(* PLC project marvel_telescope, Institute of Astronomy Onto 0.0.1 *)
(* stored: creationDateTime 2025-01-01T00:00:00.0, modificationDateTime 2025-01-01T00:00:00.0 *)

{attribute 'qualified_only'}
TYPE TelescopeNasmythPort : (UNKNOWN := 0, CHANGING := 1, POS_1 := 2, POS_2 := 3) BYTE;
END_TYPE

TYPE TelescopeProcesses : STRUCT
  {attribute 'TcHmiSymbol.Show'}
  initialize : Process;  (* Start initializing *)
  {attribute 'TcHmiSymbol.Show'}
  lock : Process;  (* Lock the cover *)
  {attribute 'TcHmiSymbol.Show'}
  unlock : Process;  (* Unlock the cover *)
  {attribute 'TcHmiSymbol.Show'}
  changeOperatingState : ChangeOperatingStateProcess;  (* Change the operating state (e.g. AUTO, MANUAL, ...) *)
  {attribute 'TcHmiSymbol.Show'}
  slewToCoordinates : PointAlphaDeltaProcess;  (* Slew to the given equatorial coordinates *)
  {attribute 'TcHmiSymbol.Show'}
  slewToAziEle : TelescopeSlewToAziEleProcess;  (* Slew to the given horizontal coordinates *)
  {attribute 'TcHmiSymbol.Show'}
  syncToCoordinates : PointAlphaDeltaProcess;  (* Sync to the given equatorial coordinates *)
  {attribute 'TcHmiSymbol.Show'}
  syncToAziEle : TelescopeSlewToAziEleProcess;  (* Sync to the given horizontal coordinates *)
  {attribute 'TcHmiSymbol.Show'}
  syncToTarget : Process;  (* Sync to the given target *)
  {attribute 'TcHmiSymbol.Show'}
  selectNasmythPort : TelescopeSelectNasmythPortProcess;  (* Select a nasmyth port *)
  {attribute 'TcHmiSymbol.Show'}
  abortSlew : Process;  (* Stop the slewing *)
  {attribute 'TcHmiSymbol.Show'}
  reset : Process;  (* Reset any errors *)
  {attribute 'TcHmiSymbol.Show'}
  powerOn : Process;  (* Power on the axes *)
  {attribute 'TcHmiSymbol.Show'}
  powerOff : Process;  (* Power off the axes *)
  {attribute 'TcHmiSymbol.Show'}
  moveKnownPosition : TelescopeMoveKnownPositionProcess;  (* Move the telescope to the given known position *)
  {attribute 'TcHmiSymbol.Show'}
  setTracking : TelescopeSetTrackingProcess;  (* Power on the axes *)
  {attribute 'TcHmiSymbol.Show'}
  moveM2 : TelescopeMoveProcess;  (* Move M2 to the given position in mm *)
  {attribute 'TcHmiSymbol.Show'}
  openCover : Process;  (* Open the telescope cover *)
  {attribute 'TcHmiSymbol.Show'}
  closeCover : Process;  (* Close the telescope cover *)
  {attribute 'TcHmiSymbol.Show'}
  pulseGuide : TelescopePulseGuideProcess;  (* Pulse guide *)
  {attribute 'TcHmiSymbol.Show'}
  guideRateAlpha : TelescopeSetRateProcess;  (* Guide right ascention rate *)
  {attribute 'TcHmiSymbol.Show'}
  guideRateDelta : TelescopeSetRateProcess;  (* Guide declination rate *)
END_STRUCT;
END_TYPE

TYPE TelescopeStatuses : STRUCT
  {attribute 'OPC.UA.DA' := '1'}
  {attribute 'OPC.UA.DA.Access' := '1'}
  {attribute 'TcHmiSymbol.Show'}
  init : InitializationStatus;
  {attribute 'OPC.UA.DA' := '1'}
  {attribute 'OPC.UA.DA.Access' := '1'}
  {attribute 'TcHmiSymbol.Show'}
  health : HealthStatus;
  {attribute 'OPC.UA.DA' := '1'}
  {attribute 'OPC.UA.DA.Access' := '1'}
  {attribute 'TcHmiSymbol.Show'}
  busy : BusyStatus;
  {attribute 'OPC.UA.DA' := '1'}
  {attribute 'OPC.UA.DA.Access' := '1'}
  {attribute 'TcHmiSymbol.Show'}
  operating : OperatingStatus;
  {attribute 'OPC.UA.DA' := '1'}
  {attribute 'OPC.UA.DA.Access' := '1'}
  {attribute 'TcHmiSymbol.Show'}
  powered : PoweredStatus;
END_STRUCT;
END_TYPE

TYPE TelescopeKnownPositionConfig : STRUCT
  {attribute 'TcHmiSymbol.Show'}
  name : STRING;  (* The name of the position (e.g. 'PARK') *)
  {attribute 'TcHmiSymbol.Show'}
  allowObserver : BOOL;  (* Can an observer switch to this position? *)
  {attribute 'TcHmiSymbol.Show'}
  azi : LREAL;  (* Azimuth in degrees *)
  {attribute 'TcHmiSymbol.Show'}
  ele : LREAL;  (* Elevation in degrees *)
  {attribute 'TcHmiSymbol.Show'}
  rot : LREAL;  (* Nasmyth rotation in degrees *)
  {attribute 'TcHmiSymbol.Show'}
  doAzi : BOOL;  (* Change the azimuth axis to the 'azi' position *)
  {attribute 'TcHmiSymbol.Show'}
  doEle : BOOL;  (* Change the elevation axis to the 'ele' position *)
  {attribute 'TcHmiSymbol.Show'}
  doRot : BOOL;  (* Change the nasmyth rotation axis to the 'rot' position *)
END_STRUCT;
END_TYPE

TYPE TelescopeKnownPositionsConfig : STRUCT
  {attribute 'TcHmiSymbol.Show'}
  position0 : TelescopeKnownPositionConfig;  (* Known position 0 *)
  {attribute 'TcHmiSymbol.Show'}
  position1 : TelescopeKnownPositionConfig;  (* Known position 1 *)
  {attribute 'TcHmiSymbol.Show'}
  position2 : TelescopeKnownPositionConfig;  (* Known position 2 *)
  {attribute 'TcHmiSymbol.Show'}
  position3 : TelescopeKnownPositionConfig;  (* Known position 3 *)
  {attribute 'TcHmiSymbol.Show'}
  position4 : TelescopeKnownPositionConfig;  (* Known position 4 *)
END_STRUCT;
END_TYPE

TYPE TelescopeConfig : STRUCT
  {attribute 'TcHmiSymbol.Show'}
  simulated : BOOL;  (* TRUE if the telescope is simulated, FALSE if not *)
  {attribute 'TcHmiSymbol.Show'}
  alpacaTelHost : STRING;  (* ASA TEL alpaca server IP address or hostname *)
  {attribute 'TcHmiSymbol.Show'}
  alpacaTelPort : UINT;  (* ASA TEL alpaca server port number *)
  {attribute 'TcHmiSymbol.Show'}
  alpacaAccHost : STRING;  (* ASA ACC alpaca server IP address or hostname *)
  {attribute 'TcHmiSymbol.Show'}
  alpacaAccPort : UINT;  (* ASA ACC alpaca server port number *)
  {attribute 'TcHmiSymbol.Show'}
  alpacaLoopTime : UINT;  (* Alpaca loop time in ms *)
  {attribute 'TcHmiSymbol.Show'}
  slewingTimeout : UINT;  (* Slewing timeout in s during pointing (both alpha/delta and azi/ele) *)
  {attribute 'TcHmiSymbol.Show'}
  knownPositions : TelescopeKnownPositionsConfig;  (* Known (predefined) positions (e.g. could be Park, Cover, Park winter, Mirror washing, ...) *)
  {attribute 'TcHmiSymbol.Show'}
  knownPositionToleranceAzi : LREAL;  (* Tolerance (in degrees) to determine if the telescope is at a known position in azi direction *)
  {attribute 'TcHmiSymbol.Show'}
  knownPositionToleranceEle : LREAL;  (* Tolerance (in degrees) to determine if the telescope is at a known position in ele direction *)
  {attribute 'TcHmiSymbol.Show'}
  knownPositionToleranceRot : LREAL;  (* Tolerance (in degrees) to determine if the telescope is at a known position in rot direction *)
  {attribute 'TcHmiSymbol.Show'}
  initSelectNasmythPort : BOOL;  (* TRUE to always select a Nasmyth port during initialization *)
  {attribute 'TcHmiSymbol.Show'}
  initSelectNasmythPortNumber : UINT;  (* Number of the nasmyth port to select during initialization *)
  {attribute 'TcHmiSymbol.Show'}
  initPower : BOOL;  (* TRUE if the power should be on or off at the end of the initialization *)
  {attribute 'TcHmiSymbol.Show'}
  initWaitForAsa : UINT;  (* Seconds to wait for the connection to the ASA PC during initialization *)
  {attribute 'TcHmiSymbol.Show'}
  nasmythSelectionTime : UINT;  (* Time in seconds to wait for M3 to switch positions (because no status can be retrieved from ASA) *)
  {attribute 'TcHmiSymbol.Show'}
  nasmythPort1Name : STRING;  (* Name of Nasmyth port 1 *)
  {attribute 'TcHmiSymbol.Show'}
  nasmythPort2Name : STRING;  (* Name of Nasmyth port 2 *)
END_STRUCT;
END_TYPE

TYPE TelescopeSlewToAziEleProcessArgs : STRUCT
  {attribute 'TcHmiSymbol.Show'}
  azimuth : LREAL;  (* Azimuth, in degrees *)
  {attribute 'TcHmiSymbol.Show'}
  elevation : LREAL;  (* Elevation, in degrees *)
END_STRUCT;
END_TYPE

TYPE TelescopePulseGuideProcessArgs : STRUCT
  {attribute 'TcHmiSymbol.Show'}
  direction : DINT;  (* Direction *)
  {attribute 'TcHmiSymbol.Show'}
  duration : DINT;  (* Duration *)
END_STRUCT;
END_TYPE

TYPE TelescopeSetRateProcessArgs : STRUCT
  {attribute 'TcHmiSymbol.Show'}
  rate : LREAL;  (* Rate (e.g. guide rate) *)
END_STRUCT;
END_TYPE

TYPE TelescopeSetTrackingProcessArgs : STRUCT
  {attribute 'TcHmiSymbol.Show'}
  tracking : BOOL;  (* Switch tracking on (TRUE) or off (FALSE) *)
END_STRUCT;
END_TYPE

TYPE TelescopeSelectNasmythPortProcessArgs : STRUCT
  {attribute 'TcHmiSymbol.Show'}
  port : UINT;  (* Port to switch to *)
END_STRUCT;
END_TYPE

TYPE TelescopeMoveKnownPositionProcessArgs : STRUCT
  {attribute 'TcHmiSymbol.Show'}
  name : STRING;  (* Name of the position to move to *)
END_STRUCT;
END_TYPE

TYPE TelescopeMoveProcessArgs : STRUCT
  {attribute 'TcHmiSymbol.Show'}
  position : LREAL;  (* New position *)
END_STRUCT;
END_TYPE

FUNCTION_BLOCK SM_Telescope
  VAR_OUTPUT
    {attribute 'OPC.UA.DA' := '1'}
    {attribute 'OPC.UA.DA.Access' := '1'}
    {attribute 'TcHmiSymbol.Show'}
    actualStatus : STRING;  (* Current status description *)
    {attribute 'TcHmiSymbol.Show'}
    {attribute 'OPC.UA.DA' := '1'}
    {attribute 'OPC.UA.DA.Access' := '1'}
    isTelConnected : BOOL;  (* True if the TEL server is connected *)
    {attribute 'TcHmiSymbol.Show'}
    {attribute 'OPC.UA.DA' := '1'}
    {attribute 'OPC.UA.DA.Access' := '1'}
    isAccConnected : BOOL;  (* True if the ACC server is connected *)
    {attribute 'TcHmiSymbol.Show'}
    {attribute 'OPC.UA.DA' := '1'}
    {attribute 'OPC.UA.DA.Access' := '1'}
    isSlewing : BOOL;  (* True if the telescope is slewing *)
    {attribute 'TcHmiSymbol.Show'}
    {attribute 'OPC.UA.DA' := '1'}
    {attribute 'OPC.UA.DA.Access' := '1'}
    isTracking : BOOL;  (* True if the telescope is tracking *)
    {attribute 'TcHmiSymbol.Show'}
    {attribute 'OPC.UA.DA' := '1'}
    {attribute 'OPC.UA.DA.Access' := '1'}
    isPulseGuiding : BOOL;  (* True if the telescope is pulse guiding *)
    {attribute 'TcHmiSymbol.Show'}
    {attribute 'OPC.UA.DA' := '1'}
    {attribute 'OPC.UA.DA.Access' := '1'}
    actAlpha : AngularPosition;  (* The actual alpha coordinate (Right Ascention) *)
    {attribute 'TcHmiSymbol.Show'}
    {attribute 'OPC.UA.DA' := '1'}
    {attribute 'OPC.UA.DA.Access' := '1'}
    actDelta : AngularPosition;  (* The actual delta coordinate (Declination) *)
    {attribute 'TcHmiSymbol.Show'}
    {attribute 'OPC.UA.DA' := '1'}
    {attribute 'OPC.UA.DA.Access' := '1'}
    actAzi : AngularPosition;  (* The actual azimuth *)
    {attribute 'TcHmiSymbol.Show'}
    {attribute 'OPC.UA.DA' := '1'}
    {attribute 'OPC.UA.DA.Access' := '1'}
    actEle : AngularPosition;  (* The actual elevation *)
    {attribute 'TcHmiSymbol.Show'}
    {attribute 'OPC.UA.DA' := '1'}
    {attribute 'OPC.UA.DA.Access' := '1'}
    actNasmythPort : TelescopeNasmythPort;  (* Actual Nasmyth port *)
    {attribute 'TcHmiSymbol.Show'}
    {attribute 'OPC.UA.DA' := '1'}
    {attribute 'OPC.UA.DA.Access' := '1'}
    actNasmythPortName : STRING;  (* Actual Nasmyth port name *)
    {attribute 'TcHmiSymbol.Show'}
    {attribute 'OPC.UA.DA' := '1'}
    {attribute 'OPC.UA.DA.Access' := '1'}
    targetAlpha : AngularPosition;  (* The target alpha coordinate (Right Ascention) *)
    {attribute 'TcHmiSymbol.Show'}
    {attribute 'OPC.UA.DA' := '1'}
    {attribute 'OPC.UA.DA.Access' := '1'}
    targetDelta : AngularPosition;  (* The target delta coordinate (Declination) *)
    {attribute 'TcHmiSymbol.Show'}
    {attribute 'OPC.UA.DA' := '1'}
    {attribute 'OPC.UA.DA.Access' := '1'}
    isAtKnownPosition : BOOL;  (* True if the telescope is at a known position *)
    {attribute 'TcHmiSymbol.Show'}
    {attribute 'OPC.UA.DA' := '1'}
    {attribute 'OPC.UA.DA.Access' := '1'}
    actualKnownPositionName : STRING;  (* Name of the known position if isAtKnownPosition is True *)
    {attribute 'TcHmiSymbol.Show'}
    stat : TelescopeStatuses;  (* Statuses of the state machine *)
    {attribute 'TcHmiSymbol.Show'}
    proc : TelescopeProcesses;  (* Processes of the state machine *)
  END_VAR
  VAR_IN_OUT
    {attribute 'TcHmiSymbol.Show'}
    {attribute 'OPC.UA.DA' := '0'}
    {attribute 'TcHmiSymbol.Hide'}
    operator_ref : OperatorStatus;  (* Shared operator status *)
    {attribute 'TcHmiSymbol.Show'}
    {attribute 'OPC.UA.DA' := '0'}
    {attribute 'TcHmiSymbol.Hide'}
    activity_ref : ActivityStatus;  (* Shared activity status *)
    {attribute 'TcHmiSymbol.Show'}
    {attribute 'OPC.UA.DA' := '0'}
    {attribute 'TcHmiSymbol.Hide'}
    services_ref : Services;  (* Shared services *)
    {attribute 'TcHmiSymbol.Show'}
    {attribute 'OPC.UA.DA' := '0'}
    {attribute 'TcHmiSymbol.Hide'}
    config_ref : TelescopeConfig;  (* Active configuration of the telescope *)
  END_VAR

            stat.health := F_HealthStatus(
    superState := NOT(stat.init = InitializationStatus.shutdown),
    isGood := (NOT(stat.init = InitializationStatus.initializingFailed)) AND (isTelConnected AND (isAccConnected AND (((proc.initialize.stat.health = HealthStatus.good) OR (proc.initialize.stat.health = HealthStatus.warning)) AND (((proc.changeOperatingState.stat.health = HealthStatus.good) OR (proc.changeOperatingState.stat.health = HealthStatus.warning)) AND (((proc.slewToCoordinates.stat.health = HealthStatus.good) OR (proc.slewToCoordinates.stat.health = HealthStatus.warning)) AND (((proc.slewToAziEle.stat.health = HealthStatus.good) OR (proc.slewToAziEle.stat.health = HealthStatus.warning)) AND (((proc.abortSlew.stat.health = HealthStatus.good) OR (proc.abortSlew.stat.health = HealthStatus.warning)) AND (((proc.powerOn.stat.health = HealthStatus.good) OR (proc.powerOn.stat.health = HealthStatus.warning)) AND (((proc.powerOff.stat.health = HealthStatus.good) OR (proc.powerOff.stat.health = HealthStatus.warning)) AND (((proc.moveKnownPosition.stat.health = HealthStatus.good) OR (proc.moveKnownPosition.stat.health = HealthStatus.warning)) AND (((proc.setTracking.stat.health = HealthStatus.good) OR (proc.setTracking.stat.health = HealthStatus.warning)) AND (((proc.moveM2.stat.health = HealthStatus.good) OR (proc.moveM2.stat.health = HealthStatus.warning)) AND (((proc.openCover.stat.health = HealthStatus.good) OR (proc.openCover.stat.health = HealthStatus.warning)) AND ((proc.closeCover.stat.health = HealthStatus.good) OR (proc.closeCover.stat.health = HealthStatus.warning))))))))))))))),
    hasWarning := (proc.initialize.stat.health = HealthStatus.warning) OR ((proc.changeOperatingState.stat.health = HealthStatus.warning) OR ((proc.slewToCoordinates.stat.health = HealthStatus.warning) OR ((proc.slewToAziEle.stat.health = HealthStatus.warning) OR ((proc.abortSlew.stat.health = HealthStatus.warning) OR ((proc.powerOn.stat.health = HealthStatus.warning) OR ((proc.powerOff.stat.health = HealthStatus.warning) OR ((proc.moveKnownPosition.stat.health = HealthStatus.warning) OR ((proc.setTracking.stat.health = HealthStatus.warning) OR ((proc.moveM2.stat.health = HealthStatus.warning) OR ((proc.openCover.stat.health = HealthStatus.warning) OR (proc.closeCover.stat.health = HealthStatus.warning))))))))))));
stat.busy := F_BusyStatus(
    superState := NOT(stat.init = InitializationStatus.shutdown),
    isBusy := (proc.initialize.stat.busy = BusyStatus.busy) OR ((proc.changeOperatingState.stat.busy = BusyStatus.busy) OR ((proc.slewToCoordinates.stat.busy = BusyStatus.busy) OR ((proc.slewToAziEle.stat.busy = BusyStatus.busy) OR ((proc.abortSlew.stat.busy = BusyStatus.busy) OR ((proc.powerOn.stat.busy = BusyStatus.busy) OR ((proc.powerOff.stat.busy = BusyStatus.busy) OR ((proc.moveKnownPosition.stat.busy = BusyStatus.busy) OR ((proc.setTracking.stat.busy = BusyStatus.busy) OR ((proc.moveM2.stat.busy = BusyStatus.busy) OR ((proc.openCover.stat.busy = BusyStatus.busy) OR (proc.closeCover.stat.busy = BusyStatus.busy))))))))))));
proc.initialize( isEnabled := (NOT(stat.init = InitializationStatus.locked)) AND ((stat.init = InitializationStatus.shutdown) OR ((stat.init = InitializationStatus.initializingFailed) OR (stat.init = InitializationStatus.initialized))) );
proc.lock( isEnabled := operator_ref = OperatorStatus.tech );
proc.unlock( isEnabled := (operator_ref = OperatorStatus.tech) AND (stat.init = InitializationStatus.locked) );
proc.changeOperatingState( isEnabled := (stat.busy = BusyStatus.idle) AND ((stat.init = InitializationStatus.initialized) AND (operator_ref = OperatorStatus.tech)) );
proc.slewToCoordinates( isEnabled := (stat.init = InitializationStatus.initialized) AND ((stat.busy = BusyStatus.idle) AND (stat.powered = PoweredStatus.enabled)) );
proc.slewToAziEle( isEnabled := (stat.init = InitializationStatus.initialized) AND ((stat.busy = BusyStatus.idle) AND (stat.powered = PoweredStatus.enabled)) );
proc.syncToCoordinates( isEnabled := (stat.init = InitializationStatus.initialized) AND ((stat.busy = BusyStatus.idle) AND (stat.powered = PoweredStatus.enabled)) );
proc.syncToAziEle( isEnabled := (stat.init = InitializationStatus.initialized) AND ((stat.busy = BusyStatus.idle) AND (stat.powered = PoweredStatus.enabled)) );
proc.syncToTarget( isEnabled := (stat.init = InitializationStatus.initialized) AND ((stat.busy = BusyStatus.idle) AND (stat.powered = PoweredStatus.enabled)) );
proc.selectNasmythPort( isEnabled := stat.init = InitializationStatus.initialized );
proc.abortSlew( isEnabled := stat.init = InitializationStatus.initialized );
proc.reset( isEnabled := (stat.busy = BusyStatus.idle) AND (stat.init = InitializationStatus.initialized) );
proc.powerOn( isEnabled := (NOT(stat.init = InitializationStatus.locked)) AND ((stat.init = InitializationStatus.initialized) AND (proc.powerOn.stat.busy = BusyStatus.idle)) );
proc.powerOff( isEnabled := (stat.init = InitializationStatus.initialized) AND (proc.powerOff.stat.busy = BusyStatus.idle) );
proc.moveKnownPosition( isEnabled := (stat.init = InitializationStatus.initialized) AND ((stat.busy = BusyStatus.idle) AND (stat.powered = PoweredStatus.enabled)) );
proc.setTracking( isEnabled := stat.init = InitializationStatus.initialized );
proc.moveM2( isEnabled := (stat.init = InitializationStatus.initialized) AND (proc.moveM2.stat.busy = BusyStatus.idle) );
proc.openCover( isEnabled := (stat.init = InitializationStatus.initialized) AND (proc.openCover.stat.busy = BusyStatus.idle) );
proc.closeCover( isEnabled := (stat.init = InitializationStatus.initialized) AND (proc.closeCover.stat.busy = BusyStatus.idle) );
proc.pulseGuide( isEnabled := (stat.init = InitializationStatus.initialized) AND (proc.pulseGuide.stat.busy = BusyStatus.idle) );
proc.guideRateAlpha( isEnabled := (stat.init = InitializationStatus.initialized) AND (proc.guideRateAlpha.stat.busy = BusyStatus.idle) );
proc.guideRateDelta( isEnabled := (stat.init = InitializationStatus.initialized) AND (proc.guideRateDelta.stat.busy = BusyStatus.idle) );

          
END_FUNCTION_BLOCK

FUNCTION_BLOCK TelescopeSlewToAziEleProcess EXTENDS BaseProcess
  VAR_INPUT
    {attribute 'OPC.UA.DA' := '1'}
    {attribute 'TcHmiSymbol.Show'}
    set : TelescopeSlewToAziEleProcessArgs;  (* Arguments to be set, before writing do_request TRUE *)
  END_VAR
  VAR_OUTPUT
    {attribute 'OPC.UA.DA' := '1'}
    {attribute 'OPC.UA.DA.Access' := '1'}
    {attribute 'TcHmiSymbol.Show'}
    get : TelescopeSlewToAziEleProcessArgs;  (* Arguments in use by the process, if do_request was accepted *)
  END_VAR

            IF do_request THEN
    do_request_result := request(
    azimuth := set.azimuth,
    elevation := set.elevation);
    do_request := FALSE;
END_IF;
SUPER^();

          

{attribute 'TcRpcEnable' := '1'}
METHOD start
  VAR_INPUT
    {attribute 'TcHmiSymbol.Show'}
    azimuth : LREAL;  (* Azimuth, in degrees *)
    {attribute 'TcHmiSymbol.Show'}
    elevation : LREAL;  (* Elevation, in degrees *)
  END_VAR
                  THIS^.get.azimuth := azimuth;
THIS^.get.elevation := elevation;
THIS^.stat.busy := BusyStatus.busy;
THIS^.stat.health := HealthStatus.good;

                
END_METHOD

{attribute 'TcRpcEnable' := '1'}
METHOD request : RequestResults
  VAR_INPUT
    {attribute 'TcHmiSymbol.Show'}
    azimuth : LREAL;  (* Azimuth, in degrees *)
    {attribute 'TcHmiSymbol.Show'}
    elevation : LREAL;  (* Elevation, in degrees *)
  END_VAR
                  IF THIS^.stat.enabled = EnabledStatus.enabled THEN
    request := RequestResults.ACCEPTED;
    THIS^.start(
        azimuth := azimuth,
        elevation := elevation);
ELSE
    request := RequestResults.REJECTED;
END_IF;

                
END_METHOD
END_FUNCTION_BLOCK

FUNCTION_BLOCK TelescopePulseGuideProcess EXTENDS BaseProcess
  VAR_INPUT
    {attribute 'OPC.UA.DA' := '1'}
    {attribute 'TcHmiSymbol.Show'}
    set : TelescopePulseGuideProcessArgs;  (* Arguments to be set, before writing do_request TRUE *)
  END_VAR
  VAR_OUTPUT
    {attribute 'OPC.UA.DA' := '1'}
    {attribute 'OPC.UA.DA.Access' := '1'}
    {attribute 'TcHmiSymbol.Show'}
    get : TelescopePulseGuideProcessArgs;  (* Arguments in use by the process, if do_request was accepted *)
  END_VAR

            IF do_request THEN
    do_request_result := request(
    direction := set.direction,
    duration := set.duration);
    do_request := FALSE;
END_IF;
SUPER^();

          

{attribute 'TcRpcEnable' := '1'}
METHOD start
  VAR_INPUT
    {attribute 'TcHmiSymbol.Show'}
    direction : DINT;  (* Direction *)
    {attribute 'TcHmiSymbol.Show'}
    duration : DINT;  (* Duration *)
  END_VAR
                  THIS^.get.direction := direction;
THIS^.get.duration := duration;
THIS^.stat.busy := BusyStatus.busy;
THIS^.stat.health := HealthStatus.good;

                
END_METHOD

{attribute 'TcRpcEnable' := '1'}
METHOD request : RequestResults
  VAR_INPUT
    {attribute 'TcHmiSymbol.Show'}
    direction : DINT;  (* Direction *)
    {attribute 'TcHmiSymbol.Show'}
    duration : DINT;  (* Duration *)
  END_VAR
                  IF THIS^.stat.enabled = EnabledStatus.enabled THEN
    request := RequestResults.ACCEPTED;
    THIS^.start(
        direction := direction,
        duration := duration);
ELSE
    request := RequestResults.REJECTED;
END_IF;

                
END_METHOD
END_FUNCTION_BLOCK

FUNCTION_BLOCK TelescopeSetRateProcess EXTENDS BaseProcess
  VAR_INPUT
    {attribute 'OPC.UA.DA' := '1'}
    {attribute 'TcHmiSymbol.Show'}
    set : TelescopeSetRateProcessArgs;  (* Arguments to be set, before writing do_request TRUE *)
  END_VAR
  VAR_OUTPUT
    {attribute 'OPC.UA.DA' := '1'}
    {attribute 'OPC.UA.DA.Access' := '1'}
    {attribute 'TcHmiSymbol.Show'}
    get : TelescopeSetRateProcessArgs;  (* Arguments in use by the process, if do_request was accepted *)
  END_VAR

            IF do_request THEN
    do_request_result := request( rate := set.rate );
    do_request := FALSE;
END_IF;
SUPER^();

          

{attribute 'TcRpcEnable' := '1'}
METHOD start
  VAR_INPUT
    {attribute 'TcHmiSymbol.Show'}
    rate : LREAL;  (* Rate (e.g. guide rate) *)
  END_VAR
                  THIS^.get.rate := rate;
THIS^.stat.busy := BusyStatus.busy;
THIS^.stat.health := HealthStatus.good;

                
END_METHOD

{attribute 'TcRpcEnable' := '1'}
METHOD request : RequestResults
  VAR_INPUT
    {attribute 'TcHmiSymbol.Show'}
    rate : LREAL;  (* Rate (e.g. guide rate) *)
  END_VAR
                  IF THIS^.stat.enabled = EnabledStatus.enabled THEN
    request := RequestResults.ACCEPTED;
    THIS^.start( rate := rate );
ELSE
    request := RequestResults.REJECTED;
END_IF;

                
END_METHOD
END_FUNCTION_BLOCK

FUNCTION_BLOCK TelescopeSetTrackingProcess EXTENDS BaseProcess
  VAR_INPUT
    {attribute 'OPC.UA.DA' := '1'}
    {attribute 'TcHmiSymbol.Show'}
    set : TelescopeSetTrackingProcessArgs;  (* Arguments to be set, before writing do_request TRUE *)
  END_VAR
  VAR_OUTPUT
    {attribute 'OPC.UA.DA' := '1'}
    {attribute 'OPC.UA.DA.Access' := '1'}
    {attribute 'TcHmiSymbol.Show'}
    get : TelescopeSetTrackingProcessArgs;  (* Arguments in use by the process, if do_request was accepted *)
  END_VAR

            IF do_request THEN
    do_request_result := request( tracking := set.tracking );
    do_request := FALSE;
END_IF;
SUPER^();

          

{attribute 'TcRpcEnable' := '1'}
METHOD start
  VAR_INPUT
    {attribute 'TcHmiSymbol.Show'}
    tracking : BOOL;  (* Switch tracking on (TRUE) or off (FALSE) *)
  END_VAR
                  THIS^.get.tracking := tracking;
THIS^.stat.busy := BusyStatus.busy;
THIS^.stat.health := HealthStatus.good;

                
END_METHOD

{attribute 'TcRpcEnable' := '1'}
METHOD request : RequestResults
  VAR_INPUT
    {attribute 'TcHmiSymbol.Show'}
    tracking : BOOL;  (* Switch tracking on (TRUE) or off (FALSE) *)
  END_VAR
                  IF THIS^.stat.enabled = EnabledStatus.enabled THEN
    request := RequestResults.ACCEPTED;
    THIS^.start( tracking := tracking );
ELSE
    request := RequestResults.REJECTED;
END_IF;

                
END_METHOD
END_FUNCTION_BLOCK

FUNCTION_BLOCK TelescopeSelectNasmythPortProcess EXTENDS BaseProcess
  VAR_INPUT
    {attribute 'OPC.UA.DA' := '1'}
    {attribute 'TcHmiSymbol.Show'}
    set : TelescopeSelectNasmythPortProcessArgs;  (* Arguments to be set, before writing do_request TRUE *)
  END_VAR
  VAR_OUTPUT
    {attribute 'OPC.UA.DA' := '1'}
    {attribute 'OPC.UA.DA.Access' := '1'}
    {attribute 'TcHmiSymbol.Show'}
    get : TelescopeSelectNasmythPortProcessArgs;  (* Arguments in use by the process, if do_request was accepted *)
  END_VAR

            IF do_request THEN
    do_request_result := request( port := set.port );
    do_request := FALSE;
END_IF;
SUPER^();

          

{attribute 'TcRpcEnable' := '1'}
METHOD start
  VAR_INPUT
    {attribute 'TcHmiSymbol.Show'}
    port : UINT;  (* Port to switch to *)
  END_VAR
                  THIS^.get.port := port;
THIS^.stat.busy := BusyStatus.busy;
THIS^.stat.health := HealthStatus.good;

                
END_METHOD

{attribute 'TcRpcEnable' := '1'}
METHOD request : RequestResults
  VAR_INPUT
    {attribute 'TcHmiSymbol.Show'}
    port : UINT;  (* Port to switch to *)
  END_VAR
                  IF THIS^.stat.enabled = EnabledStatus.enabled THEN
    request := RequestResults.ACCEPTED;
    THIS^.start( port := port );
ELSE
    request := RequestResults.REJECTED;
END_IF;

                
END_METHOD
END_FUNCTION_BLOCK

FUNCTION_BLOCK TelescopeMoveKnownPositionProcess EXTENDS BaseProcess
  VAR_INPUT
    {attribute 'OPC.UA.DA' := '1'}
    {attribute 'TcHmiSymbol.Show'}
    set : TelescopeMoveKnownPositionProcessArgs;  (* Arguments to be set, before writing do_request TRUE *)
  END_VAR
  VAR_OUTPUT
    {attribute 'OPC.UA.DA' := '1'}
    {attribute 'OPC.UA.DA.Access' := '1'}
    {attribute 'TcHmiSymbol.Show'}
    get : TelescopeMoveKnownPositionProcessArgs;  (* Arguments in use by the process, if do_request was accepted *)
  END_VAR

            IF do_request THEN
    do_request_result := request( name := set.name );
    do_request := FALSE;
END_IF;
SUPER^();

          

{attribute 'TcRpcEnable' := '1'}
METHOD start
  VAR_INPUT
    {attribute 'TcHmiSymbol.Show'}
    name : STRING;  (* Name of the position to move to *)
  END_VAR
                  THIS^.get.name := name;
THIS^.stat.busy := BusyStatus.busy;
THIS^.stat.health := HealthStatus.good;

                
END_METHOD

{attribute 'TcRpcEnable' := '1'}
METHOD request : RequestResults
  VAR_INPUT
    {attribute 'TcHmiSymbol.Show'}
    name : STRING;  (* Name of the position to move to *)
  END_VAR
                  IF THIS^.stat.enabled = EnabledStatus.enabled THEN
    request := RequestResults.ACCEPTED;
    THIS^.start( name := name );
ELSE
    request := RequestResults.REJECTED;
END_IF;

                
END_METHOD
END_FUNCTION_BLOCK

FUNCTION_BLOCK TelescopeMoveProcess EXTENDS BaseProcess
  VAR_INPUT
    {attribute 'OPC.UA.DA' := '1'}
    {attribute 'TcHmiSymbol.Show'}
    set : TelescopeMoveProcessArgs;  (* Arguments to be set, before writing do_request TRUE *)
  END_VAR
  VAR_OUTPUT
    {attribute 'OPC.UA.DA' := '1'}
    {attribute 'OPC.UA.DA.Access' := '1'}
    {attribute 'TcHmiSymbol.Show'}
    get : TelescopeMoveProcessArgs;  (* Arguments in use by the process, if do_request was accepted *)
  END_VAR

            IF do_request THEN
    do_request_result := request( position := set.position );
    do_request := FALSE;
END_IF;
SUPER^();

          

{attribute 'TcRpcEnable' := '1'}
METHOD start
  VAR_INPUT
    {attribute 'TcHmiSymbol.Show'}
    position : LREAL;  (* New position *)
  END_VAR
                  THIS^.get.position := position;
THIS^.stat.busy := BusyStatus.busy;
THIS^.stat.health := HealthStatus.good;

                
END_METHOD

{attribute 'TcRpcEnable' := '1'}
METHOD request : RequestResults
  VAR_INPUT
    {attribute 'TcHmiSymbol.Show'}
    position : LREAL;  (* New position *)
  END_VAR
                  IF THIS^.stat.enabled = EnabledStatus.enabled THEN
    request := RequestResults.ACCEPTED;
    THIS^.start( position := position );
ELSE
    request := RequestResults.REJECTED;
END_IF;

                
END_METHOD
END_FUNCTION_BLOCK
